FUNCTION Convert_REAL_TO_BOOL : BOOL
VAR_INPUT
	in : REAL;
	out : REFERENCE TO BOOL;
END_VAR
VAR
	converted : BOOL;
END_VAR

converted := REAL_TO_BOOL(in);

IF (BOOL_TO_REAL(converted) <> in) THEN
	RETURN;
END_IF

out := converted;
Convert_REAL_TO_BOOL := TRUE;

END_FUNCTION

(* stored: Version 1.1.0.1, ProductVersion 3.1.4024.12
   POU Convert_REAL_TO_BOOL: Id {404ab3c5-0597-4dee-9d9b-3cfa72342579}, SpecialFunc None *)
